(* CODESYS project mainV2_RECOVERED_2025-03-20T13-50-34.project

Project tree, tasks and I/O mapping:
  Device : 751-9301 WAGO Compact Controller 100, WAGO, order no. 751-9301, version 6.3.1.5
    application Application
      libraries: Standard, 3.5.18.0 (System); SysSocket Implementation, * (System); SysSocket, * (System); UDP, * (3S - Smart Software Solutions GmbH); SysSocket2, * (System)
      task MainTask (cyclic, interval t#50ms, priority 15) calls PLC_PRG
      task EtherCAT_Task (cyclic, interval t#4ms, priority 1) calls nothing
      function MotorAngleToCounts [ST]
      function block MotorDriver [ST]: speedToCounts, calibrateMotor, distanceFromCenter
      function block UDPReciever [ST]: UDPDecoder
      program PLC_PRG [ST]
      function block PID [ST]
      function UDPDecoder [ST]
      function block PlatformSimulator [ST]
      function block UDPReciever2 [ST]: UDPDecoder
      function block ComputeMotorAngles [ST]
    Serial
      COM1 : COM1, WAGO, version 0.0.0.19
    Compact_Controller_100_Onboard_IO : Compact Controller 100 Onboard IO, WAGO, version 0.0.1.4
        unmapped channels: X12.DI, X13.PT1+/X13.PT1-, X13.PT2+/X13.PT2-, X14.AI1, X14.AI2, X5.DO, X6.AO1, X6.AO2
    EtherCAT_Master : EtherCAT Master, CODESYS, version 4.7.0.0
        settings: SlaveAutoRestart = True; NetworkName = 'ethX2'; NetworkName = "ethX2"; SrcAddress1 = 48; SrcAddress2 = 3730183477; EnableSecondAdapter = 2B3
  pou UDPReciver [ST]
  function block UDPReciever2 [ST]
*)

// Device/Application/PLC_PRG
PROGRAM PLC_PRG
VAR
	noe: UDPReciever;
	noeAnnet: INT;
	endaAnnet: UDINT_IN_BYTES;
	endaNoeAnnet: UDPReciever2;
	enMotorDrive: MotorDriver;
END_VAR

noeAnnet := noeAnnet + 1;
noe.port := 5;
noe.ipAddress := 2093683980;
endaNoeAnnet.xStart := TRUE;
endaNoeAnnet.sIpAddress := '192.68.50.50';

END_PROGRAM

// Device/Application/UDPReciever
FUNCTION_BLOCK UDPReciever
VAR_INPUT
    ipAddress : UDINT;
    port      : UINT;
END_VAR
VAR_OUTPUT
	floatArray : ARRAY [0..66] OF REAL;
END_VAR
VAR
    connected    : BOOL := TRUE;
    hSocket      : POINTER TO BYTE := 0;
    stAddress    : SOCKADDRESS;
    buffer       : ARRAY [0..263] OF BYTE;
    bytesReceived: LINT;
    bPrevEnable  : BOOL := FALSE;
    i            : INT;
    hexPacket    : STRING := '';
END_VAR


IF hSocket = 0 THEN
	//Må finne ut hva som skal være i steden for buffer[0] (Pointer to runtime system error code)
    hSocket := SysSockCreate(SOCKET_AF_INET, SOCKET_DGRAM, SOCKET_IPPROTO_UDP, buffer[0]);

    //Setter socket adressa
    stAddress.sin_family := SOCKET_AF_INET;
    stAddress.sin_port := SysSockHtons(port);
    stAddress.sin_addr.ulAddr := ipAddress;
    
	FOR i := 0 TO 7 DO
         stAddress.sin_zero[i] := 0;
    END_FOR;
	
    (*Binder socketen*)
    SysSockBind(hSocket, ADR(stAddress), SIZEOF(stAddress));
END_IF;

(*Mottar UDP socketet*)
IF connected THEN
    bytesReceived := SysSockRecvFrom(hSocket, ADR(buffer), SIZEOF(buffer), 0, ADR(stAddress), SIZEOF(stAddress), 0);
	floatArray := UDPDecoder(buffer);
END_IF;

METHOD UDPDecoder : ARRAY[0..66] OF REAL
VAR_INPUT
	buffer : ARRAY [0..263] OF BYTE;
END_VAR
VAR
	numberToMakeBinary: DWORD;
	binaryHexAsInt: ARRAY[0..65] OF ARRAY[0..31] OF BOOL;
 	i: INT;
	j: INT;
	k: INT;
	counter: INT := 0;
	sign: INT;
	exponent: REAL;
	mantissa: REAL;
END_VAR
counter := 0;
FOR i := 0 TO 65 DO
    	numberToMakeBinary := 0;
    	FOR k := 0 TO 3 DO
		(*Gjør om byten til binary*)
        	numberToMakeBinary := SHL(numberToMakeBinary, 8) OR (buffer[4*i + (3 - k)]);
       	counter := counter + 1;
    	END_FOR;

    	FOR j := 0 TO 31 DO
        	binaryHexAsInt[i][j] := (numberToMakeBinary AND SHL(1, 31 - j)) <> 0;
    	END_FOR;
	(*Finner ut hvilket fortegn flyttallet har*)
    	IF NOT binaryHexAsInt[i][0] THEN
		sign := 0;
	ELSE
		sign := 1;
	END_IF
	(*Regner ut eksponenten*)
    	exponent := 0;
    	FOR j := 1 TO 8 DO
        	IF binaryHexAsInt[i][j] THEN
            		exponent := exponent + EXPT(2, 8 - j);
       	END_IF;
    	END_FOR;
	    exponent := exponent - 127;
		(*Regner ut mantissaen*)
	    mantissa := 0.0;
	    FOR j := 9 TO 31 DO
	        IF binaryHexAsInt[i][j] THEN
            		mantissa := mantissa + EXPT(2, 8 - j);
       	END_IF;
    	END_FOR;
	(*Finner tallverdien*)
    	UDPDecoder[i] := EXPT(-1, DINT_TO_REAL(sign)) * (1.0 + mantissa) * EXPT(2, exponent);
END_FOR;
END_METHOD

END_FUNCTION_BLOCK

// Device/Application/UDPDecoder
FUNCTION UDPDecoder : ARRAY[0..66] OF REAL
VAR_INPUT
	buffer : ARRAY [0..263] OF BYTE;
END_VAR
VAR
	numberToMakeBinary: DWORD;
	binaryHexAsInt: ARRAY[0..65] OF ARRAY[0..31] OF BOOL;
 	i: INT;
	j: INT;
	k: INT;
	counter: INT := 0;
	sign: INT;
	exponent: REAL;
	mantissa: REAL;
END_VAR

counter := 0;
FOR i := 0 TO 65 DO
    	numberToMakeBinary := 0;
    	FOR k := 0 TO 3 DO
		(*Gjør om byten til binary*)
        	numberToMakeBinary := SHL(numberToMakeBinary, 8) OR (buffer[4*i + (3 - k)]);
       	counter := counter + 1;
    	END_FOR;

    	FOR j := 0 TO 31 DO
        	binaryHexAsInt[i][j] := (numberToMakeBinary AND SHL(1, 31 - j)) <> 0;
    	END_FOR;
	(*Finner ut hvilket fortegn flyttallet har*)
    	IF NOT binaryHexAsInt[i][0] THEN
		sign := 0;
	ELSE
		sign := 1;
	END_IF
	(*Regner ut eksponenten*)
    	exponent := 0;
    	FOR j := 1 TO 8 DO
        	IF binaryHexAsInt[i][j] THEN
            		exponent := exponent + EXPT(2, 8 - j);
       	END_IF;
    	END_FOR;
	    exponent := exponent - 127;
		(*Regner ut mantissaen*)
	    mantissa := 0.0;
	    FOR j := 9 TO 31 DO
	        IF binaryHexAsInt[i][j] THEN
            		mantissa := mantissa + EXPT(2, 8 - j);
       	END_IF;
    	END_FOR;
	(*Finner tallverdien*)
    	UDPDecoder[i] := EXPT(-1, DINT_TO_REAL(sign)) * (1.0 + mantissa) * EXPT(2, exponent);
END_FOR;

END_FUNCTION

// UDPReciever2
FUNCTION_BLOCK UDPReciever2
VAR_INPUT
    xStart: BOOL;
    sIpAddress: STRING;
    wPort: WORD;
    aDataSend: STRING;
END_VAR

VAR_OUTPUT
    aDataRec: STRING;
    xiSentBytes:  __XINT;
    xiRecBytes:  __XINT;
    createResult: syssocket_interfaces.RTS_IEC_RESULT;
    connectResult: syssocket_interfaces.RTS_IEC_RESULT;
    ieSendResult: syssocket_interfaces.RTS_IEC_RESULT;
    ieRecResult: syssocket_interfaces.RTS_IEC_RESULT;
    ieCloseResult: syssocket_interfaces.RTS_IEC_RESULT;
END_VAR

VAR
    step: INT := 1;
    socketId: syssocket_interfaces.RTS_IEC_HANDLE;
    ipAddress: syssocket.SOCKADDRESS;
END_VAR

syssocket.SysSockInetAddr(ipAddress, ADR(sIpAddress));
ipAddress.sin_family := syssocket.SOCKET_AF_INET;
ipAddress.sin_port := syssocket.SysSockHtons(wPort);

CASE step OF 
    1:
        IF xStart THEN 
            socketId := syssocket.SysSockCreate(syssocket.SOCKET_AF_INET, syssocket.SOCKET_STREAM, syssocket.SOCKET_IPPROTO_IP, ADR(createResult));
            IF socketId = syssocket_interfaces.RTS_INVALID_HANDLE THEN 
                xStart := FALSE;
                step := 1;
            ELSE 
                step := 2;    
            END_IF
        END_IF

    2:
        connectResult := syssocket.SysSockConnect(socketId, ADR(ipAddress), SIZEOF(ipAddress));
        step := 3;

    3:
        xiSentBytes := syssocket.SysSockSend(socketId, ADR(aDataSend), SIZEOF(aDataSend), 1, ADR(ieSendResult));
        step := 4;

    4:
        xiRecBytes := syssocket.SysSockRecv(socketId, ADR(aDataRec), SIZEOF(aDataRec), 1, ADR(ieRecResult));
        step := 5;

    5:
        ieCloseResult := syssocket.SysSockClose(socketId);
        xStart := FALSE;
        step := 1;
END_CASE

END_FUNCTION_BLOCK

// Device/Application/UDPReciever2
FUNCTION_BLOCK UDPReciever2
VAR_INPUT
    xStart: BOOL;
    sIpAddress: STRING;
    wPort: WORD;
    aDataSend: STRING;
END_VAR

VAR_OUTPUT
    aDataRec: STRING;
    xiSentBytes:  __XINT;
    xiRecBytes:  __XINT;
    createResult: syssocket_interfaces.RTS_IEC_RESULT;
    connectResult: syssocket_interfaces.RTS_IEC_RESULT;
    ieSendResult: syssocket_interfaces.RTS_IEC_RESULT;
    ieRecResult: syssocket_interfaces.RTS_IEC_RESULT;
    ieCloseResult: syssocket_interfaces.RTS_IEC_RESULT;
END_VAR

VAR
    step: INT := 1;
    socketId: syssocket_interfaces.RTS_IEC_HANDLE;
    ipAddress: syssocket.SOCKADDRESS;
END_VAR

//Tror ikke denne linja gjør noe
syssocket.SysSockInetAddr(sIpAddress, ADR(sIpAddress));
//Setter port familien og porten
ipAddress.sin_family := syssocket.SOCKET_AF_INET;
ipAddress.sin_port := syssocket.SysSockHtons(wPort);

CASE step OF 
    1:
		//Setter opp socketen
        IF xStart THEN 
            socketId := syssocket.SysSockCreate(syssocket.SOCKET_AF_INET, syssocket.SOCKET_STREAM, syssocket.SOCKET_IPPROTO_IP, ADR(createResult));
            IF socketId = syssocket_interfaces.RTS_INVALID_HANDLE THEN 
                xStart := FALSE;
                step := 1;
            ELSE
				//Går videre til neste steg hvis socketen blir satt opp
                step := 2;    
            END_IF
        END_IF

    2:
        connectResult := syssocket.SysSockConnect(socketId, ADR(ipAddress), SIZEOF(ipAddress));
        step := 3;

    3:
		//Sender bytes
        xiSentBytes := syssocket.SysSockSend(socketId, ADR(aDataSend), SIZEOF(aDataSend), 1, ADR(ieSendResult));
        step := 4;

    4:
		//Mottar bytes
        xiRecBytes := syssocket.SysSockRecv(socketId, ADR(aDataRec), SIZEOF(aDataRec), 1, ADR(ieRecResult));
        step := 5;

    5:
		//Lukker socketen og starter på nytt
        ieCloseResult := syssocket.SysSockClose(socketId);
        xStart := FALSE;
        step := 1;
END_CASE

METHOD UDPDecoder : ARRAY[0..66] OF REAL
VAR_INPUT
	buffer : ARRAY [0..263] OF BYTE;
END_VAR
VAR
	numberToMakeBinary: DWORD;
	binaryHexAsInt: ARRAY[0..65] OF ARRAY[0..31] OF BOOL;
 	i: INT;
	j: INT;
	k: INT;
	counter: INT := 0;
	sign: INT;
	exponent: REAL;
	mantissa: REAL;
END_VAR
counter := 0;
FOR i := 0 TO 65 DO
    	numberToMakeBinary := 0;
    	FOR k := 0 TO 3 DO
		(*Gjør om byten til binary*)
        	numberToMakeBinary := SHL(numberToMakeBinary, 8) OR (buffer[4*i + (3 - k)]);
       	counter := counter + 1;
    	END_FOR;

    	FOR j := 0 TO 31 DO
        	binaryHexAsInt[i][j] := (numberToMakeBinary AND SHL(1, 31 - j)) <> 0;
    	END_FOR;
	(*Finner ut hvilket fortegn flyttallet har*)
    	IF NOT binaryHexAsInt[i][0] THEN
		sign := 0;
	ELSE
		sign := 1;
	END_IF
	(*Regner ut eksponenten*)
    	exponent := 0;
    	FOR j := 1 TO 8 DO
        	IF binaryHexAsInt[i][j] THEN
            		exponent := exponent + EXPT(2, 8 - j);
       	END_IF;
    	END_FOR;
	    exponent := exponent - 127;
		(*Regner ut mantissaen*)
	    mantissa := 0.0;
	    FOR j := 9 TO 31 DO
	        IF binaryHexAsInt[i][j] THEN
            		mantissa := mantissa + EXPT(2, 8 - j);
       	END_IF;
    	END_FOR;
	(*Finner tallverdien*)
    	UDPDecoder[i] := EXPT(-1, DINT_TO_REAL(sign)) * (1.0 + mantissa) * EXPT(2, exponent);
END_FOR;
END_METHOD

END_FUNCTION_BLOCK

// Device/Application/MotorDriver
FUNCTION_BLOCK MotorDriver
VAR_INPUT
	wantedMotor0: LREAL;
	wantedMotor1: LREAL;
	wantedMotor2: LREAL;
	endSwitchMotor0: BOOL;
	endSwitchMotor1: BOOL;
	endSwitchMotor2: BOOL;
	currentPosition0: DINT;
	currentPosition1: DINT;
	currentPosition2: DINT;
	calibrating: BOOL;
END_VAR
VAR_OUTPUT
	speedMotor0: DINT;
	speedMotor1: DINT;
	speedMotor2: DINT;
END_VAR
VAR
	endSwitchPosition: INT := 0;
	calibrated0: BOOL := FALSE;
	calibrated1: BOOL := FALSE;
	calibrated2: BOOL := FALSE;
	prevEndSwitch0: BOOL := TRUE;
	prevEndSwitch1: BOOL := TRUE;
	prevEndSwitch2: BOOL := TRUE;
	PIDMotor0: PID;
	PIDMotor1: PID;
	PIDMotor2: PID;
	motor0ToCenter: LREAL := 0;
	motor1ToCenter: LREAL := 0;
	motor2ToCenter: LREAL := 0;
	integralEffectMotorToCenter: LREAL := 0.01;
END_VAR

IF calibrating THEN
	//Kjører kalibreringsfunksjonen på motorene
	IF NOT calibrated0 THEN
		IF endSwitchMotor0 AND prevEndSwitch0 THEN
			speedMotor0 := calibrateMotor(endSwitchMotor0);
			prevEndSwitch0 := endSwitchMotor0;
		ELSIF NOT endSwitchMotor0 THEN
			speedMotor0 := calibrateMotor(endSwitchMotor0);
			prevEndSwitch0 := endSwitchMotor0;
		ELSIF NOT prevEndSwitch0 AND endSwitchMotor0 THEN
			calibrated0 := TRUE;
		END_IF
	END_IF
	
	IF NOT calibrated1 THEN
		IF endSwitchMotor1 AND prevEndSwitch1 THEN
			speedMotor1 := calibrateMotor(endSwitchMotor1);
			prevEndSwitch1 := endSwitchMotor1;
		ELSIF NOT endSwitchMotor1 THEN
			speedMotor1 := calibrateMotor(endSwitchMotor1);
			prevEndSwitch1 := endSwitchMotor1;
		ELSIF NOT prevEndSwitch1 AND endSwitchMotor1 THEN
			calibrated1 := TRUE;
		END_IF
	END_IF
	
	IF NOT calibrated2 THEN
		IF endSwitchMotor2 AND prevEndSwitch2 THEN
			speedMotor2 := calibrateMotor(endSwitchMotor2);
			prevEndSwitch2 := endSwitchMotor2;
		ELSIF NOT endSwitchMotor1 THEN
			speedMotor2 := calibrateMotor(endSwitchMotor2);
			prevEndSwitch2 := endSwitchMotor2;
		ELSIF NOT prevEndSwitch2 AND endSwitchMotor2 THEN
			calibrated2 := TRUE;
		END_IF
	END_IF
	
	IF calibrated0 AND calibrated1 AND calibrated2 THEN
		calibrating := FALSE;
		PIDMotor0.kP := 1.2;
		PIDMotor0.kI := 0.001;
		PIDMotor0.kD := 2.5;
		PIDMotor1.kP := 1.2;
		PIDMotor1.kI := 0.001;
		PIDMotor1.kD := 2.5;
		PIDMotor2.kP := 1.2;
		PIDMotor2.kI := 0.001;
		PIDMotor2.kD := 2.5;
		calibrated0 := FALSE;
		calibrated1 := FALSE;
		calibrated2 := FALSE;
		prevEndSwitch0 := TRUE;
		prevEndSwitch1 := TRUE;
		prevEndSwitch2 := TRUE;
	END_IF
ELSE
	//Kjører bare hvis ingen av end switchene er inne
	//Er en end switch inne er noe feil
	IF endSwitchMotor0 AND endSwitchMotor1 AND endSwitchMotor2 THEN
		//Endrer ønska posisjon til å dra motorene litt mot midten for å bli klar til nytt sprang
		//pi/80000 gir antallet radianer den skal endres med
		wantedMotor0 := wantedMotor0 - motor0ToCenter * (3.1415926/80000);
		wantedMotor1 := wantedMotor1 - motor1ToCenter * (3.1415926/80000);
		wantedMotor2 := wantedMotor2 - motor2ToCenter * (3.1415926/80000);
		
		//Kjører PID kontrolleren på motorene
		PIDMotor0.currentPos := currentPosition0;
		PIDMotor0.wantedPos := wantedMotor0;
		PIDMotor1.currentPos := currentPosition1;
		PIDMotor1.wantedPos := wantedMotor1;
		PIDMotor2.currentPos := currentPosition2;
		PIDMotor2.wantedPos := wantedMotor2;
		
		//Setter hastigheta
		speedMotor0 := speedToCounts(PIDMotor0.sum + motor0ToCenter, currentPosition0);
		speedMotor1 := speedToCounts(PIDMotor1.sum + motor1ToCenter, currentPosition1);
		speedMotor2 := speedToCounts(PIDMotor2.sum + motor2ToCenter, currentPosition2);
		
		//Lager en integraleffekt som drar motorene sakte mot midten
		motor0ToCenter := motor0ToCenter + distanceFromCenter(currentPosition0) * integralEffectMotorToCenter;
		motor1ToCenter := motor1ToCenter + distanceFromCenter(currentPosition1) * integralEffectMotorToCenter;
		motor2ToCenter := motor2ToCenter + distanceFromCenter(currentPosition2) * integralEffectMotorToCenter;
		
		//Slutter å dra mot midten om den er nært nok midten
		IF currentPosition0 > 35000 AND currentPosition0 < 45000 THEN
			motor0ToCenter := 0;
		END_IF
		IF currentPosition1 > 35000 AND currentPosition1 < 45000 THEN
			motor1ToCenter := 0;
		END_IF
		IF currentPosition2 > 35000 AND currentPosition2 < 45000 THEN
			motor2ToCenter := 0;
		END_IF
		
		
	ELSE
		//Skrur av alle motorene om en endswitch plutselig er inne
		speedMotor0 := 0;
		speedMotor1 := 0;
		speedMotor2 := 0;
	END_IF
END_IF

METHOD speedToCounts : DINT
VAR_INPUT
	wantedSpeed: LREAL;
	currentPosition: DINT;
END_VAR
VAR
	outputSpeed: DINT;
	maxOutput: DINT := 3600;
	maxExpectedWanted: LREAL := 10;
	//Maks og min position i motor counts
	minPosition: DINT := 100;
	maxPosition: DINT := 80000;
END_VAR
//Etter 3600 i hastighet får man overspeed error. Gjetting på at maksimal wanted speed er omtrent 10
outputSpeed := REAL_TO_DINT((maxOutput/maxExpectedWanted) * wantedSpeed);
IF outputSpeed > maxOutput THEN
	outputSpeed := maxOutput;
ELSIF outputSpeed < -maxOutput THEN
	outputSpeed := -maxOutput;
END_IF

//Setter farta til 0 hvis den prøver å bevege seg forbi maksimalposisjonene
IF currentPosition >= maxPosition AND outputSpeed > 0 THEN
	outputSpeed := 0;
ELSIF currentPosition <= maxPosition AND outputSpeed < 0 THEN
	outputSpeed := 0;
END_IF

speedToCounts := outputSpeed;
END_METHOD

METHOD calibrateMotor : DINT
VAR_INPUT
	endSwitch: BOOL;
END_VAR
VAR
	calibrationSpeed: DINT;
END_VAR
calibrateMotor := -calibrationSpeed;
END_METHOD

METHOD distanceFromCenter : LREAL
VAR_INPUT
	currentPos: DINT;
END_VAR
VAR
	prevTime: TIME;
	deltaTime: REAL;
	centerPos: DINT := 40000;
END_VAR
//Ikke helt stuereint å gange med deltaTime her, men det er for at deltaTime skal påvirke det løpende integralet
deltaTime := TIME_TO_REAL(TIME() - prevTime);
distanceFromCenter := (centerPos - currentPos) * deltaTime;
prevTime := TIME();
END_METHOD

END_FUNCTION_BLOCK

// Device/Application/PID
FUNCTION_BLOCK PID
VAR_INPUT
	kP: REAL;
	kI: REAL;
	kD: REAL;
	wantedPos: LREAL;
	currentPos: DINT;
END_VAR
VAR_OUTPUT
	sum: LREAL;
END_VAR
VAR
	prevError: LREAL;
	integral: LREAL;
	lastTime: TIME := TIME();
	deltaTime: REAL;
	error: LREAL; 
END_VAR

deltaTime := TIME_TO_REAL(TIME() - lastTime);
lastTime := TIME();
wantedPos := MotorAngleToCounts(wantedPos);
error := wantedPos - currentPos;

sum := kP * error;
sum := sum + kD * (error - prevError) * deltaTime;
sum := sum + kI * integral * deltaTime;

prevError := error;
integral := integral + error;

END_FUNCTION_BLOCK

// Device/Application/MotorAngleToCounts
FUNCTION MotorAngleToCounts : DINT
VAR_INPUT
	wantedMotorAngle: LREAL;
END_VAR
VAR
	motorCountsPerRound: REAL := 160000;
	pi: REAL := 3.1415926;
	tempVar: DINT;
END_VAR

MotorAngleToCounts := LREAL_TO_DINT((wantedMotorAngle * motorCountsPerRound)/(2*pi));

END_FUNCTION

// Device/Application/PlatformSimulator
FUNCTION_BLOCK PlatformSimulator
VAR_INPUT
	motorInput1  :  DINT;
   	motorInput2  :  DINT;
   	motorInput3  :  DINT;
END_VAR
VAR_OUTPUT
	platformPitch : REAL;
    platformRoll : REAL;
	limitSwitch1 : BOOL;
	limitSwitch2 : BOOL;
	limitSwitch3 : BOOL;
END_VAR
VAR
	motorAngle1 : REAL;
	motorAngle2 : REAL;
    motorAngle3 : REAL;
    p1 : REAL;
    p2 : REAL;
    p3 : REAL;
END_VAR

(*Tar inn motor countsene og ganger det med 1/1 rotasjon (160000) og ganger med 2pi FOR å få det til radianer*)
motorAngle1 := motorInput1 * 0.0000392699;
motorAngle2 := motorInput2 * 0.0000392699;
motorAngle3 := motorInput3 * 0.0000392699;

(*Sjekker om limit switchene er trykka inn*)
limitSwitch1 := NOT((motorAngle1 > (350 * 0.01745328627) AND motorAngle1 < (359 * 0.01745328627)));
limitSwitch2 := NOT((motorAngle2 > (350 * 0.01745328627) AND motorAngle2 < (359 * 0.01745328627)));
limitSwitch3 := NOT((motorAngle3 > (350 * 0.01745328627) AND motorAngle3 < (359 * 0.01745328627)));

(*Regner ut høyde over platformen*)
p1 := 0.08 * (1 - COS(motorAngle1));
p2 := 0.08 * (1 - COS(motorAngle2));
p3 := 0.08 * (1 - COS(motorAngle3));

(*Regner ut pitch og roll på platforma*)
platformPitch := ATAN((p2 - ((p3 + p1) / 2)) / ((1.75 * SQRT(3)) / 2));

platformRoll := ATAN((p3 - p1) / 1.75);

END_FUNCTION_BLOCK

// Device/Application/ComputeMotorAngles
FUNCTION_BLOCK ComputeMotorAngles
VAR_INPUT
	roll : LREAL;
	pitch : LREAL;
END_VAR
VAR_OUTPUT
	angle0 : LREAL;
	angle1 : LREAL;
	angle2 : LREAL;

	didBound : BOOL;
END_VAR
VAR
	l : LREAL := 1.75;
	delta : LREAL := 0.08;
	s0 : LREAL := 1.0;
	s1 : LREAL := 1.0;

	tmpVar0 : LREAL;
	tmpVar1 : LREAL;

	p0 : LREAL;
	p1 : LREAL;
	p2 : LREAL;
END_VAR

tmpVar0 := l / 2 * ATAN(roll);
p1 := delta + tmpVar0;
p0 := delta - tmpVar0;

tmpVar1 := (l * SQRT(3) / 2) * ATAN(-pitch) / 2;
p2 := delta - tmpVar1;

p0 := p0 + tmpVar1;
p1 := p1 + tmpVar1;

p0 := -1.0 * (p0 - delta) / delta;
p1 := -1.0 * (p1 - delta) / delta;
p2 := -1.0 * (p2 - delta) / delta;

didBound := FALSE;

IF (p0 > 1.0) THEN
	p0 := 1.0;
	didBound := TRUE;
ELSIF (p0 < -1.0) THEN
	p0 := -1.0;
	didBound := TRUE;
END_IF


IF (p1 > 1.0) THEN
	p1 := 1.0;
	didBound := TRUE;
ELSIF (p1 < -1.0) THEN
	p1 := -1.0;
	didBound := TRUE;
END_IF

IF (p2 > 1.0) THEN
	p2 := 1.0;
	didBound := TRUE;
ELSIF (p2 < -1.0) THEN
	p2 := -1.0;
	didBound := TRUE;
END_IF

angle0 := ACOS(p0);
angle2 := ACOS(p1);
angle1 := ACOS(p2);

END_FUNCTION_BLOCK
